PROGRAM PRG_04_AirValveAnalytics
VAR	
	AirValve							: ARRAY [1..6] OF Valve2Cmd2FB;
	
	{attribute 'OPC.UA.DA' := '0'}
	{attribute 'OPC.UA.DA.Access' := '1'}			// read only
	{attribute 'OPC.UA.DA.StructuredType' := '1'}
	AirValveStruct01					: ValveTravelTime_DataModel;
	
	{attribute 'OPC.UA.DA' := '0'}
	{attribute 'OPC.UA.DA.Access' := '1'}			// read only
	{attribute 'OPC.UA.DA.StructuredType' := '1'}
	AirValveStruct02					: ValveTravelTime_DataModel;
	

	AirValveStruct03						: ValveTravelTime_DataModel;
	AirValveStruct04						: ValveTravelTime_DataModel;
	

END_VAR


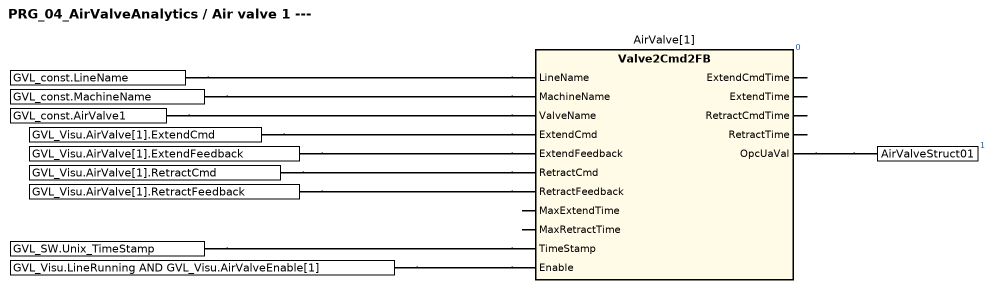
// PAGE Air valve 1 ---
AirValve[1](
    LineName := GVL_const.LineName,
    MachineName := GVL_const.MachineName,
    ValveName := GVL_const.AirValve1,
    ExtendCmd := GVL_Visu.AirValve[1].ExtendCmd,
    ExtendFeedback := GVL_Visu.AirValve[1].ExtendFeedback,
    RetractCmd := GVL_Visu.AirValve[1].RetractCmd,
    RetractFeedback := GVL_Visu.AirValve[1].RetractFeedback,
    TimeStamp := GVL_SW.Unix_TimeStamp,
    Enable := GVL_Visu.LineRunning AND GVL_Visu.AirValveEnable[1]); // Valve2Cmd2FB
AirValveStruct01 := AirValve[1].OpcUaVal;

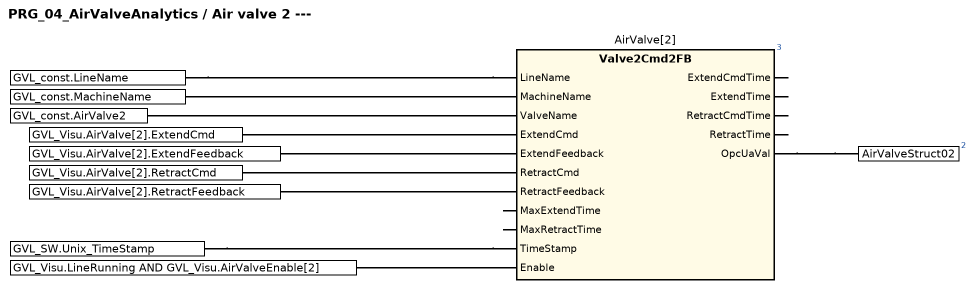
// PAGE Air valve 2 ---
AirValveStruct02 := AirValve[2].OpcUaVal;
AirValve[2](
    LineName := GVL_const.LineName,
    MachineName := GVL_const.MachineName,
    ValveName := GVL_const.AirValve2,
    ExtendCmd := GVL_Visu.AirValve[2].ExtendCmd,
    ExtendFeedback := GVL_Visu.AirValve[2].ExtendFeedback,
    RetractCmd := GVL_Visu.AirValve[2].RetractCmd,
    RetractFeedback := GVL_Visu.AirValve[2].RetractFeedback,
    TimeStamp := GVL_SW.Unix_TimeStamp,
    Enable := GVL_Visu.LineRunning AND GVL_Visu.AirValveEnable[2]); // Valve2Cmd2FB

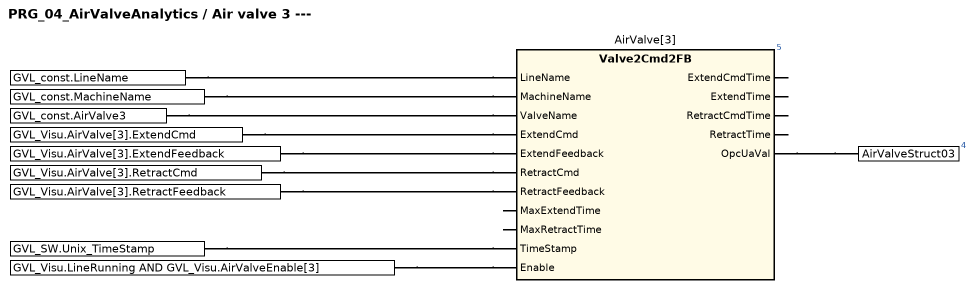
// PAGE Air valve 3 ---
AirValveStruct03 := AirValve[3].OpcUaVal;
AirValve[3](
    LineName := GVL_const.LineName,
    MachineName := GVL_const.MachineName,
    ValveName := GVL_const.AirValve3,
    ExtendCmd := GVL_Visu.AirValve[3].ExtendCmd,
    ExtendFeedback := GVL_Visu.AirValve[3].ExtendFeedback,
    RetractCmd := GVL_Visu.AirValve[3].RetractCmd,
    RetractFeedback := GVL_Visu.AirValve[3].RetractFeedback,
    TimeStamp := GVL_SW.Unix_TimeStamp,
    Enable := GVL_Visu.LineRunning AND GVL_Visu.AirValveEnable[3]); // Valve2Cmd2FB

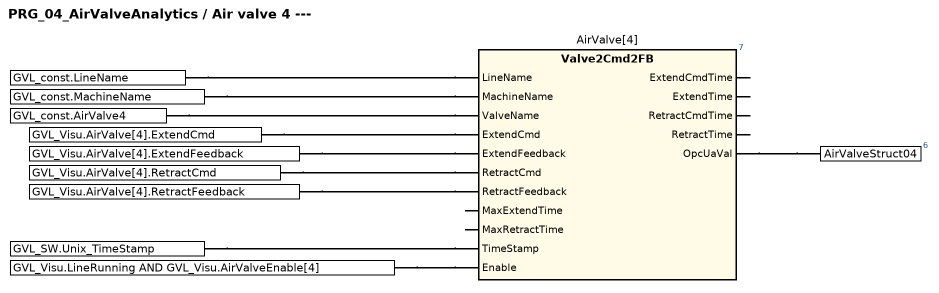
// PAGE Air valve 4 ---
AirValveStruct04 := AirValve[4].OpcUaVal;
AirValve[4](
    LineName := GVL_const.LineName,
    MachineName := GVL_const.MachineName,
    ValveName := GVL_const.AirValve4,
    ExtendCmd := GVL_Visu.AirValve[4].ExtendCmd,
    ExtendFeedback := GVL_Visu.AirValve[4].ExtendFeedback,
    RetractCmd := GVL_Visu.AirValve[4].RetractCmd,
    RetractFeedback := GVL_Visu.AirValve[4].RetractFeedback,
    TimeStamp := GVL_SW.Unix_TimeStamp,
    Enable := GVL_Visu.LineRunning AND GVL_Visu.AirValveEnable[4]); // Valve2Cmd2FB

END_PROGRAM

(* stored: Version 1.1.0.1, ProductVersion 3.1.4024.15
   POU PRG_04_AirValveAnalytics: Id {2d34a1e7-0ed3-47a9-952f-f80601f3c6db}, SpecialFunc None *)
